// TIA Portal V20 export
TYPE "typeEm1MonitoringJobInterface"
// stored: Access Published, Namespace Unit1
   STRUCT
      busyRewind { ExternalWritable := 'False'} : Bool;
      busyLinkChg { ExternalWritable := 'False'} : Bool;
      doneRewind { ExternalWritable := 'False'} : Bool;
      doneLinkChg { ExternalWritable := 'False'} : Bool;
   END_STRUCT;
END_TYPE
